{attribute addProperty BoxType "EL3122--0000"}
{attribute addProperty Id "ChannelAT %I*ARRAY[0..2] OF Channel_A23A2BD94860WcStateAT %I*WcState_98A4DF7520.250InfoDataAT %I*InfoData_BC63D37F80100"}
{attribute addProperty CRC "4081952094"}
{attribute addProperty SizeInBites "130"}
{attribute addProperty SizeInBytes "16.25"}
TYPE EL3122_C619ACF8 :
STRUCT
	{attribute addProperty Name "Channel"}
	Channel : ARRAY[0..2] OF Channel_A23A2BD9;
	{attribute addProperty Name "WcState"}
	WcState : WcState_98A4DF75;
	{attribute addProperty Name "InfoData"}
	InfoData : InfoData_BC63D37F;
END_STRUCT
END_TYPE

(* stored: Version 1.2.0.0, ProductVersion 3.1.4024.9
   DUT EL3122_C619ACF8: Id {ce8be940-b719-4ff8-b53e-eb24f384e21a} *)
